FUNCTION_BLOCK HMatrixReverseAccessor EXTENDS MatrixAccessor
VAR_INPUT
END_VAR
VAR_OUTPUT
END_VAR
VAR
END_VAR

//Total number of columns in this matrix
PROPERTY PUBLIC Cols : UINT
GET
IF NOT __ISVALIDREF(M_) THEN
	Cols := 0;
	LogWarning('%s Attempted Cols access using uninitialized Matrix Accessor');
ELSE
	Cols := M_.Rows;
END_IF
END_GET
END_PROPERTY

METHOD PUBLIC GetI : LREAL
VAR_INPUT
	I : UINT;
END_VAR
VAR
	ThisR : UINT;
	ThisC : UINT;
END_VAR
IC2RC(I,Cols,Row => ThisR, Col => ThisC);

IF (ThisR < 3 AND ThisC < 3) OR ThisR = ThisC THEN
	//Transpose the R part or the diagonal (no mod)
	GetI := SUPER^.GetI(I);
ELSE
	//do not transpose the other parts (they will get negated isntead)
	getI := -1 * SUPER^.GetI(I);
END_IF
END_METHOD

METHOD PUBLIC Init
VAR_INPUT
	M : REFERENCE TO HMatrix;
END_VAR
Init_(M);
END_METHOD

//Total number of rows in this matrix
PROPERTY PUBLIC Rows : UINT
GET
IF NOT __ISVALIDREF(M_) THEN
	Rows := 0;
	LogWarning('%s Attempted Rows access using uninitialized Matrix Accessor');
ELSE
	Rows := M_.Cols;
END_IF
END_GET
END_PROPERTY

METHOD PUBLIC SetI : BOOL
VAR_INPUT
	I : UINT;
	Val : LREAL;
END_VAR
VAR
	ThisR : UINT;
	ThisC : UINT;
END_VAR
IC2RC(I,Cols,Row => ThisR, Col => ThisC);

IF (ThisR < 3 AND ThisC < 3) OR ThisR = ThisC THEN
	//Transpose the R part or the diagonal (no mod)
	SetI := SUPER^.SetI(I,Val);
ELSE
	//do not transpose the other parts (they will get negated isntead)
	SetI := SUPER^.SetI(I,-1*Val);
END_IF
END_METHOD

METHOD PROTECTED This2Parent : UINT
VAR_INPUT
	Index : UINT;
END_VAR
VAR
	ThisR : UINT;
	ThisC : UINT;
END_VAR
IF NOT __ISVALIDREF(M_) THEN
	LogWarning('%s Attempted This2Parent calculation using uninitialized Matrix Accessor');
	This2Parent := 0;
	RETURN;
END_IF

IC2RC(Index,Cols,Row => ThisR, Col => ThisC);

IF (ThisR < 3 AND ThisC < 3) OR ThisR = ThisC THEN
	//Transpose the R part or the diagonal (no mod)
	This2Parent := RCC2I(ThisC,ThisR,M_.Cols);
ELSE
	//do not transpose the other parts (they will get negated isntead)
	This2Parent := RCC2I(ThisR,ThisC,M_.Cols);
END_IF
END_METHOD

END_FUNCTION_BLOCK

(* stored: Version 1.1.0.1, ProductVersion 3.1.4024.9
   POU HMatrixReverseAccessor: Id {33fefcdb-926f-0c7b-0261-3622c514816a}, SpecialFunc None
   Folder Initializers: Id {fbb3bcae-92bb-0187-2edb-c1e9f4b2ebea}
   Folder Overrides: Id {445fad87-5c75-0ee0-13b4-cd3564957305}
   Property Cols: Id {38bf019a-6d1a-0ddb-0b0c-32af462480f2}
   Get Get: Id {4ccd7500-5ee9-0a33-1c6f-5e05d86f5daa}
   Method GetI: Id {2bbfe692-2637-051a-3d40-ef8411d338fd}
   Method Init: Id {4b571c14-7ad7-0359-3c92-05a5516b311e}
   Property Rows: Id {d623675a-c4f7-0845-3b45-1858fde00567}
   Get Get: Id {700ca6bc-e747-0ddc-28b5-8570744aacd2}
   Method SetI: Id {06e47383-69e0-0f9a-2195-4f3ea2ae21e6}
   Method This2Parent: Id {050b5be5-0368-003f-2fdb-79ca646ab29d} *)
